// TwinCAT 3 PLC project StageCore
// Title: StageCore
// Company: _
// Author: Krystian Lis et al.
// ProjectVersion: 3.2.0
// ProgramVersion: 3.1.4026.16
// libraries:
//   Tc2_Math, * (Beckhoff Automation GmbH)
//   Tc2_Standard, * (Beckhoff Automation GmbH)
//   Tc2_System, * (Beckhoff Automation GmbH)
//   Tc2_Utilities, * (Beckhoff Automation GmbH)
// project tree:
//   Arg/Args/BOOL/ IArgToIBoolArg.TcPOU (not stored), BoolArg.TcPOU (not stored), I_BoolArg.TcIO (not stored)
//   Arg/Args/REAL/ IArgToIRealtArg.TcPOU (not stored), RealArg.TcPOU, I_RealArg.TcIO
//   Arg/Args/DWORD/ IArgToIDwordArg.TcPOU (not stored), DwordArg.TcPOU (not stored), I_DwordArg.TcIO
//   Arg/ ICompToIArg.TcPOU (not stored), IArgToIComp.TcPOU (not stored), I_Arg.TcIO (not stored)
//   Broadcast/Helpers/ GetSignal.TcPOU, GetReceiver.TcPOU (not stored)
//   Broadcast/Receiver/ AbstractReceiver.TcPOU (not stored), ICompToIRec.TcPOU, I_Receiver.TcIO, I_ReceiverNode.TcIO, Receiver.TcPOU (not stored)
//   Broadcast/Signal/ ICompToISignal.TcPOU, I_SignalEmit.TcIO (not stored), I_Signal.TcIO (not stored), I_SignalNode.TcIO, Signal.TcPOU (not stored)
//   Broadcast/Sys/Helpers/ _BroadcastDefragment.TcPOU, _BroadcastGetBestFit.TcPOU (not stored), _Emit.TcPOU, _Pair.TcPOU (not stored), _RegSignal.TcPOU (not stored), _Unpair.TcPOU
//   Broadcast/Sys/Structs/ _BroadcastStruct.TcDUT (not stored), _BroadcastUnion.TcDUT
//   Broadcast/Sys/ _Broadcast.TcGVL
//   Callable/ I_Callable.TcIO (not stored)
//   Dbg/ DebugInfo.TcPOU (not stored), DebugMsg.TcPOU, DebugStr.TcPOU (not stored), I_Debug.TcIO (not stored), _DebugInfo.TcDUT (not stored), _Debug.TcGVL (not stored)
//   Entity/Core/ Component.TcPOU, I_Component.TcIO, GetOwnerFromRaw.TcPOU, I_RawComponent.TcIO, I_Entity.TcIO (not stored), GetNextEntity.TcPOU, GetPrevEntity.TcPOU
//   Entity/Core/Scope/ EntityEnd.TcPOU (not stored), EntityExtend.TcPOU (not stored), EntityStart.TcPOU
//   Entity/Sys/ _EntityState.TcDUT, _Ec.TcGVL (not stored)
//   Entity/Sys/_Helpers/ _EntityEnd.TcPOU (not stored), _EntityExtend.TcPOU, _EntityStart.TcPOU, _RegisterComponent.TcPOU (not stored)
//   Entity/Sys/_Itf/ I_ComponentNode.TcIO (not stored), I_EntityNode.TcIO
//   Iter/ Iter.TcPOU
//   Result/Error/ Err.TcGVL, GenericResult.TcGVL (not stored)
//   Result/ IsErr.TcPOU (not stored), IsNone.TcPOU, IsOk.TcPOU (not stored), IsFail.TcPOU (not stored), IsSome.TcPOU (not stored), IsEnd.TcPOU, Result.TcDUT, ResultToStr.TcPOU
//   Runtime/Execute/ Execute.TcPOU (not stored), I_Execute.TcIO (not stored), I_ExecuteNode.TcIO
//   Runtime/Init/ Init.TcPOU, I_InitNode.TcIO, I_Init.TcIO (not stored)
//   Runtime/ Runtime.TcPOU, _Runtime.TcGVL (not stored)
//   State/_Buffer/ _StateBuffer.TcPOU (not stored)
//   State/Helpers/ GetStateManager.TcPOU, GetState.TcPOU
//   State/_Machine/ _StateMachine.TcPOU (not stored)
//   State/Manager/ ICompToIStateMgr.TcPOU (not stored), I_StateManager.TcIO, StateManager.TcPOU (not stored)
//   State/State/ ICompToIState.TcPOU, I_State.TcIO (not stored), I_StateInternal.TcIO (not stored), I_StateAdapter.TcIO (not stored), State.TcPOU (not stored)
//   Strings/Alias/ Ch.TcDUT, Str.TcDUT (not stored)
//   Strings/Strb/ I_Strb.TcIO (not stored), Strb.TcPOU (not stored)
//   Strings/Strf/ Strf.TcPOU (not stored)
//   Tags/Casts/ IArgToITag.TcPOU (not stored), ICompToITag.TcPOU, ICompToITagged.TcPOU
//   Tags/Helpers/ GetTag.TcPOU (not stored), GetTagOption.TcPOU, HasTagOption.TcPOU (not stored), HasTag.TcPOU, MatchPath.TcPOU
//   Tags/ I_Tag.TcIO, I_TagCmp.TcIO (not stored), I_Tagged.TcIO, TagBase.TcPOU (not stored), TagCmp.TcPOU, TagPath.TcPOU (not stored), Tag.TcPOU (not stored)
//   Tasks/Worker/Base/ Worker.TcPOU (not stored), I_Worker.TcIO
//   Tasks/Worker/ LoopWorker.TcPOU (not stored), BlockingWorker.TcPOU (not stored)
//   Tasks/TaskNode/ I_JobNode.TcIO, I_JobNodeInternal.TcIO, Job.TcPOU (not stored)
//   Tasks/ TaskState.TcDUT
//   Tasks/Job/ I_Job.TcIO (not stored)
//   _/ Param.TcGVL
// (motion and I/O tree: see PLC project stageutils)
// real-time tasks:
//   TASK Example: cycle T#10ms, priority 20, ADS port 350
//   TASK Test: cycle T#10ms, priority 21, ADS port 351
//   TASK VISU_TASK: cycle T#200000us, priority 30, ADS port 352

// ---- Broadcast/Sys/Structs/_BroadcastUnion.TcDUT
TYPE INTERNAL  _BroadcastUnion :
UNION
	iSignal		: I_SignalNode;
	iReceiver	: I_ReceiverNode;
END_UNION
END_TYPE

// ---- Entity/Sys/_EntityState.TcDUT
{attribute 'qualified_only'}
{attribute 'strict'}
TYPE INTERNAL _EntityState :
(
	Unregistered,
	Registered,
	Completed
);
END_TYPE

// ---- Result/Result.TcDUT
// Alias for INT values.
// | Result >= 1 - Ok/Success
// | Result = 0 - None
// | Result <=- 1 - Error
TYPE Result : INT; END_TYPE

// ---- Strings/Alias/Ch.TcDUT
// Alias for STRING(1) values.
TYPE Ch : STRING(1); END_TYPE

// ---- Tasks/TaskState.TcDUT
{attribute 'qualified_only'}
{attribute 'strict'}
TYPE TaskState :
(
	Error,
	Idle,
	Ready,
	Running,
	Aborted,
	Completed
) BYTE := Idle;
END_TYPE

// ---- Broadcast/Sys/_Broadcast.TcGVL
{attribute 'qualified_only'}
VAR_GLOBAL INTERNAL
	{attribute 'ExpandFully'} 
	entry				: ARRAY[1..Param.RECEIVER_CAP] OF _BroadcastStruct;
	iSignal				: ARRAY[1..Param.SIGNAL_CAP] OF I_SignalNode;
	iFirst				: I_SignalNode;
	nRecLen				: UDINT;
	nSignalLen			: UDINT;
END_VAR

// ---- Result/Error/Err.TcGVL
{attribute 'qualified_only'}
VAR_GLOBAL CONSTANT
	Itf0			: Result := -2; // Null Interface 
	Str0			: Result := -3; // Empty String
	ItfEq			: Result := -4; // Interfaces are equal
	NoMatch			: Result := -5; // No match
	Ptr0			: Result := -6; // Null Pointer
	InvRef			: Result := -7; // Invalid reference
	Ovf				: Result := -8; // Overflow/Out of bounds
	Udf				: Result := -9; // Undefined
	Idx				: Result := -10; // Index error
	TcLib			: Result := -11; // Error caused by TwinCAT libraries
	InfLoop			: Result := -12; // Potential infinity loop
	IncArg			: Result := -13; // Incorrect input argument
	Init			: Result := -14; // Initialisation error
	NotFound		: Result := -15; // Item not found
	InvItf			: Result := -16; // Invalid interface
	End				: Result := -17; // End of collection
END_VAR

// ---- _/Param.TcGVL
{attribute 'qualified_only'}
// DO NOT SET ANY OF THE CAP PARAMETERS TO 0 OR LARGER THAN MAX DINT!!!
VAR_GLOBAL CONSTANT
	DEBUGMSG_CAP	: UDINT(1..16#7FFFFFFF) := 10; // Max number of debug messages.
	DEBUGSTR_CAP	: UDINT(1..16#7FFFFFFF) := 500; // Max number of debug strings.
	
	SIGNAL_CAP		: UDINT(1..16#7FFFFFFF) := 20; // Max number of signals.
	RECEIVER_CAP	: UDINT(1..16#7FFFFFFF) := 100; // Max number of signal-receiver pairings.
END_VAR

// ---- Arg/Args/REAL/I_RealArg.TcIO
(*
A broadcastable wrapper for a `REAL` value. 
*)
INTERFACE I_RealArg EXTENDS I_Arg

(*
Reads the internal value.
*)
PROPERTY Get : REAL
GET
END_GET
END_PROPERTY

(*
Returns TRUE if the value is mutable.
*)
PROPERTY IsMut : BOOL
GET
END_GET
END_PROPERTY

(*
Modifies the internal value.  
Returns:
- `Ok` - Upon successful modification.
- `Error` - If mutability is disabled.
*)
METHOD Set : Result
VAR_INPUT
	newVal		: REAL;
END_VAR
END_METHOD

END_INTERFACE

// ---- Arg/Args/DWORD/I_DwordArg.TcIO
(*
A broadcastable wrapper for a `DWORD` value. 
*)
INTERFACE I_DwordArg EXTENDS I_Arg

(*
Reads the internal value.
*)
PROPERTY Get : DWORD
GET
END_GET
END_PROPERTY

(*
Returns TRUE if the value is mutable.
*)
PROPERTY IsMut : BOOL
GET
END_GET
END_PROPERTY

(*
Modifies the internal value.  
Returns:
- `Ok` - Upon successful modification.
- `Error` - If mutability is disabled.
*)
METHOD Set : Result
VAR_INPUT
	newVal		: DWORD;
END_VAR
END_METHOD

END_INTERFACE

// ---- Broadcast/Receiver/I_Receiver.TcIO
(*
Represents a receiver in the Broadcast system. Implements the necessary methods for receiving events and pairing signals.
Can be casted to `I_Component`.
*)
INTERFACE I_Receiver EXTENDS I_ReceiverNode, I_Tagged

END_INTERFACE

// ---- Broadcast/Receiver/I_ReceiverNode.TcIO
INTERFACE INTERNAL I_ReceiverNode EXTENDS I_Debug

METHOD INTERNAL Receive
VAR_INPUT
	iArg			: I_Arg;
END_VAR
END_METHOD

END_INTERFACE

// ---- Broadcast/Signal/I_SignalNode.TcIO
INTERFACE INTERNAL I_SignalNode EXTENDS I_Debug

PROPERTY INTERNAL _End : UDINT
GET
END_GET
SET
END_SET
END_PROPERTY

PROPERTY INTERNAL _Id : UDINT
GET
END_GET
END_PROPERTY

PROPERTY INTERNAL _Size : UDINT
GET
END_GET
SET
END_SET
END_PROPERTY

PROPERTY INTERNAL _Start : UDINT
GET
END_GET
SET
END_SET
END_PROPERTY

END_INTERFACE

// ---- Entity/Core/I_Component.TcIO
(*
Stores raw I_RawComponent value and additional metadata.
*)
INTERFACE I_Component EXTENDS I_ComponentNode

(*
Returns parent Entity.
*)
PROPERTY Entity : I_Entity
GET
END_GET
END_PROPERTY

(*
Returns raw I_RawComponent pointer.
*)
PROPERTY Raw : I_RawComponent
GET
END_GET
END_PROPERTY

END_INTERFACE

// ---- Entity/Core/I_RawComponent.TcIO
(*
Represents a component in the Entity-Component system.  
Can be cast to other interfaces for extended functionality and interaction.
*)
INTERFACE I_RawComponent EXTENDS __SYSTEM.IQueryInterface, I_Debug

END_INTERFACE

// ---- Entity/Sys/_Itf/I_EntityNode.TcIO
INTERFACE INTERNAL I_EntityNode EXTENDS I_Debug

PROPERTY INTERNAL _AsIEntity : I_Entity
GET
END_GET
END_PROPERTY

PROPERTY INTERNAL _FirstComp : I_ComponentNode
GET
END_GET
SET
END_SET
END_PROPERTY

PROPERTY INTERNAL _LastComp : I_ComponentNode
GET
END_GET
SET
END_SET
END_PROPERTY

PROPERTY INTERNAL _Next : I_EntityNode
GET
END_GET
SET
END_SET
END_PROPERTY

PROPERTY INTERNAL _Prev : I_EntityNode
GET
END_GET
SET
END_SET
END_PROPERTY

PROPERTY INTERNAL _Size : UDINT
GET
END_GET
SET
END_SET
END_PROPERTY

PROPERTY INTERNAL _State : _EntityState
GET
END_GET
SET
END_SET
END_PROPERTY

(*
Description: Retrieves a previous component before the inputted one or last component if referenced value is 0.
Returns:
- Ok - Returns upon success, updates referenced value with new component.
- Err.InvRef - Invalid output reference.
- Err.ItfEq - Provided interface pointer doesn't belong to the queried entity. Nulls reference.
- Err.NotFound - The entity doesn't contain any components. Nulls reference.
- Err.End - No more components. Nulls reference.
*)
METHOD GetNextComp : Result
VAR_INPUT
	iOut		: REFERENCE TO I_Component;
END_VAR
END_METHOD

(*
Description: Retrieves a previous component before the inputted one or last component if referenced value is 0.
Returns:
- Ok - Returns upon success, updates referenced value with new component.
- Err.InvRef - Invalid output reference.
- Err.ItfEq - Provided interface pointer doesn't belong to the queried entity. Nulls reference.
- Err.NotFound - The entity doesn't contain any components. Nulls reference.
- Err.End - No more components. Nulls reference.
*)
METHOD GetPrevComp : Result
VAR_INPUT
	iOut		: REFERENCE TO I_Component;
END_VAR
END_METHOD

(*
Provides the size of the entity, indicating the number of components it manages.  
Note: For internal logic purposes, this value is incremented by one beyond the actual component count.
*)
PROPERTY Size : UDINT
GET
END_GET
END_PROPERTY

END_INTERFACE

// ---- Runtime/Execute/I_ExecuteNode.TcIO
INTERFACE INTERNAL I_ExecuteNode EXTENDS I_Debug;

METHOD INTERNAL Attach : Result
VAR_INPUT
	iExecute		: I_ExecuteNode;
END_VAR
END_METHOD

METHOD INTERNAL Exe
VAR_OUTPUT
	iNext: I_ExecuteNode;
END_VAR
END_METHOD

PROPERTY INTERNAL State : Result
GET
END_GET
SET
END_SET
END_PROPERTY

END_INTERFACE

// ---- Runtime/Init/I_InitNode.TcIO
INTERFACE INTERNAL I_InitNode EXTENDS I_Debug;

METHOD INTERNAL Attach : Result
VAR_INPUT
	iInit		: I_InitNode;
END_VAR
END_METHOD

METHOD INTERNAL Init
VAR_OUTPUT
	iNext: I_InitNode;
END_VAR
END_METHOD

PROPERTY INTERNAL State : Result
GET
END_GET
SET
END_SET
END_PROPERTY

END_INTERFACE

// ---- State/Manager/I_StateManager.TcIO
(*
Can be casted to `I_Component`.
Manages the lifecycle and transitions of states within an entity.  
Supports queuing state change requests, triggering state transitions, and broadcasting state change events.  
Adds a `_stateChangeEvent` Signal to the owning `I_Entity` during initialization, enabling external components to listen for state changes.
*)
INTERFACE I_StateManager EXTENDS I_Debug, I_RawComponent

(*
Retrieves the currently active state managed by the state manager.
*)
PROPERTY Current : I_State
GET
END_GET
END_PROPERTY

(*
Returns the entity that owns this state.
*)
PROPERTY Owner : I_Entity
GET
END_GET
END_PROPERTY

(*
Retrieves the state that is queued to become active next, but has not yet transitioned.
*)
PROPERTY Pretender : I_State
GET
END_GET
END_PROPERTY

(*
Retrieves the last active state prior to the current one.
*)
PROPERTY Previous : I_State
GET
END_GET
END_PROPERTY

(*
Queues a request to transition to a specified state.  

Returns:
- `Ok` - If the state change request is successfully queued.
- `Err.Itf0` - If the provided state interface is invalid.
- `Err.NoMatch` - If the state does not belong to the same entity.
- `Err.IncArg` - If the state is already in the queue.
*)
METHOD Request : Result
VAR_INPUT
	iState		: I_State;
END_VAR
END_METHOD

END_INTERFACE

// ---- Tags/I_Tag.TcIO
(*
An identifier that uses reflection to generate a unique symbol path.
It simplifies the path by removing project, PLC, and tag segments.
Can be casted to `I_Arg` and `I_Component`.
Example:
- Reflection: proj.plc.MAIN.functionBlock[*]._tag
- Path: MAIN.functionBlock.5
*)
INTERFACE I_Tag EXTENDS I_Debug, I_Component, I_Arg

// Read address path without Option segment.
PROPERTY Id : Str
GET
END_GET
END_PROPERTY

// Modify or read the optional segment.
PROPERTY Option : Str
GET
END_GET
END_PROPERTY

END_INTERFACE

// ---- Tags/I_Tagged.TcIO
(*
This component contains readable `I_Tag`.
Can be casted to `I_Component`.
*)
INTERFACE I_Tagged EXTENDS I_RawComponent

PROPERTY Tag : I_Tag
GET
END_GET
END_PROPERTY

END_INTERFACE

// ---- Tasks/Worker/Base/I_Worker.TcIO
INTERFACE I_Worker EXTENDS I_Debug

METHOD Defer : Result
VAR_INPUT
    iJob : I_JobNode;
END_VAR
END_METHOD

METHOD Dequeue : Result
VAR_INPUT
	iJob: I_JobNode;
END_VAR
END_METHOD

METHOD Enqueue : Result
VAR_INPUT
	iJob: I_JobNode;
END_VAR
END_METHOD

PROPERTY First : I_JobNode
GET
END_GET
END_PROPERTY

END_INTERFACE

// ---- Tasks/TaskNode/I_JobNode.TcIO
INTERFACE I_JobNode EXTENDS I_JobNodeInternal

END_INTERFACE

// ---- Tasks/TaskNode/I_JobNodeInternal.TcIO
INTERFACE INTERNAL I_JobNodeInternal EXTENDS I_Debug

PROPERTY INTERNAL _Next : I_JobNode
GET
END_GET
SET
END_SET
END_PROPERTY

PROPERTY INTERNAL _Prev : I_JobNode
GET
END_GET
SET
END_SET
END_PROPERTY

METHOD INTERNAL _Reset
VAR_INPUT
END_VAR
END_METHOD

METHOD INTERNAL _Run
VAR_INPUT
END_VAR
END_METHOD

PROPERTY State : TaskState
GET
END_GET
END_PROPERTY

PROPERTY Worker : I_Worker
GET
END_GET
END_PROPERTY

END_INTERFACE

// ---- Runtime/Init/Init.TcPOU
(*
Allows registration of FB implementing `I_Init`. 
*)
FUNCTION_BLOCK FINAL Init IMPLEMENTS I_InitNode, I_Debug
VAR
	_iInit			: I_Init;
	_iNext			: I_InitNode;
	_nState			: Result;
	_nPhase			: INT;
END_VAR

METHOD INTERNAL Attach : Result
VAR_INPUT
	iInit			: I_InitNode;
END_VAR
VAR
	_iThis			: I_InitNode := THIS^;
END_VAR
IF iInit = 0 THEN
	DebugMsg(0, Tc2_Standard.CONCAT(__POUNAME(), ': Itf = 0!'));
	RETURN;
END_IF

IF _iThis <> _Runtime.iLastInit THEN
	DebugMsg(THIS^, Tc2_Standard.CONCAT(__POUNAME(), ': Is not the last node!'));
	RETURN;
END_IF

IF IsSome(iInit.state) THEN
	DebugMsg(iInit, Tc2_Standard.CONCAT(__POUNAME(), ': Has already been added!'));
	RETURN;
END_IF

_Runtime.iLastInit := iInit;
_iNext := iInit;
END_METHOD

//FB_Init is always available implicitly and it is used primarily for initialization.
//The return value is not evaluated. For a specific influence, you can also declare the
//methods explicitly and provide additional code there with the standard initialization
//code. You can evaluate the return value.
{attribute 'hide'}
METHOD FB_Init: BOOL
VAR_INPUT
    bInitRetains: BOOL; // TRUE: the retain variables are initialized (reset warm / reset cold)
    bInCopyCode: BOOL;  // TRUE: the instance will be copied to the copy code afterward (online change)
	
	iInit			: I_Init;
END_VAR
IF IsSome(_nState) THEN
	RETURN;
END_IF

IF (_iInit := iInit) = 0 THEN
	_nState := Err.Itf0;
	DebugMsg(THIS^, Tc2_Standard.CONCAT(__POUNAME(), ': Itf = 0!'));
	RETURN;
END_IF



IF _Runtime.iLastInit <> 0 THEN
	IF IsErr(_Runtime.iLastInit.Attach(THIS^), nOut => _nState) THEN
		DebugMsg(THIS^, Tc2_Standard.CONCAT(__POUNAME(), ': Error Inside!'));
	END_IF
ELSE
	_Runtime.iFirstInit := THIS^;
	_Runtime.iLastInit := THIS^;
	_nState := Ok;
END_IF
END_METHOD

METHOD INTERNAL Init
VAR_OUTPUT
	iNext: I_InitNode;
END_VAR
_iInit.Init(_nPhase);
iNext := _iNext;
END_METHOD

PROPERTY Phase : INT
GET
Phase := _nPhase;
END_GET
SET
_nPhase := Phase;
END_SET
END_PROPERTY

PROPERTY INTERNAL State : Result
GET
State := _nState;
END_GET
SET
IF IsNone(_nState) THEN
	_nState := State;
END_IF
END_SET
END_PROPERTY

END_FUNCTION_BLOCK

// ---- Dbg/DebugMsg.TcPOU
(*
Logs a debug message as a string tied to a `I_Debug` interface for inspection and troubleshooting within the IDE.
*)
FUNCTION DebugMsg
VAR_INPUT
	iDebug			: I_Debug;
	sInfo			: Str;
END_VAR

_Debug.nErrorNumber := _Debug.nErrorNumber + 1;

IF _Debug.nLastMsg < Param.DEBUGMSG_CAP THEN
	_Debug.nLastMsg := _Debug.nLastMsg + 1;
ELSE
	_Debug.nLastMsg := 1;
END_IF

_Debug.debugMsg[_Debug.nLastMsg].iDebug := iDebug;
_Debug.debugMsg[_Debug.nLastMsg].sInfo := sInfo;

END_FUNCTION

// ---- Result/IsNone.TcPOU
// Return TRUE if the value is None.
// Optionally carries the value over to nOut for further processing.
FUNCTION IsNone : BOOL
VAR_INPUT
    nIn : Result; // Result variable to check for None
END_VAR
VAR_OUTPUT
    nOut : Result; // Carries the input value for further use
END_VAR

IsNone := nIn = 0;
nOut := nIn;

END_FUNCTION

// ---- Arg/Args/REAL/RealArg.TcPOU
(*
A broadcastable wrapper for a `REAL` value. 
*)
FUNCTION_BLOCK RealArg IMPLEMENTS I_RealArg
VAR
	_val			: REAL;
	_bMut			: BOOL := FALSE;
END_VAR

(*
Enables external modification of the internal value.
*)
METHOD AllowMut
_bMut := TRUE;
END_METHOD

(*
Disables external modification of the internal value.
*)
METHOD BlockMut
_bMut := FALSE;
END_METHOD

//FB_Init is always available implicitly and it is used primarily for initialization.
//The return value is not evaluated. For a specific influence, you can also declare the
//methods explicitly and provide additional code there with the standard initialization
//code. You can evaluate the return value.
{attribute 'hide'}
METHOD FB_Init: BOOL
VAR_INPUT
    bInitRetains: BOOL; // TRUE: the retain variables are initialized (reset warm / reset cold)
    bInCopyCode: BOOL;  // TRUE: the instance will be copied to the copy code afterward (online change)   

	initVal		: REAL;
END_VAR
_val := initVal;
END_METHOD

(*
Reads the internal value.
*)
PROPERTY Get : REAL
GET
Get := _val;
END_GET
END_PROPERTY

(*
Returns TRUE if the value is mutable.
*)
PROPERTY IsMut : BOOL
GET
IsMut := _bMut;
END_GET
END_PROPERTY

(*
Directly modifies the internal value, bypassing any mutability restrictions.
*)
METHOD OpSet : I_Arg
VAR_INPUT
	newVal		: REAL;
END_VAR
_val := newVal;
OpSet := THIS^;
END_METHOD

(*
Modifies the internal value.  
Returns:
- `Ok` - Upon successful modification.
- `Error` - If mutability is disabled.
*)
METHOD Set : Result
VAR_INPUT
	newVal		: REAL;
END_VAR
IF _bMut THEN
	_val := newVal;
	Set := Ok;
ELSE
	Set := Error;
END_IF
END_METHOD

END_FUNCTION_BLOCK

// ---- Broadcast/Helpers/GetSignal.TcPOU
(*
Searches an `I_Entity` for a `I_Signal` component matching provided id pattern.
Result:
- Ok - Returns `I_Signal`.
- Err.NotFound - Returns null.
- Err.InvRef - Returns null.
- Err.Itf0 - Returns null, incorrect interface.
*)
FUNCTION GetSignal : Result
VAR_INPUT
	iEntity		: I_Entity;
	sTagId		: Str;
	iOut		: REFERENCE TO I_Signal;
END_VAR
VAR
	_iComp		: I_Component;
	cmp			: TagCmp;
END_VAR

IF iEntity = 0 THEN
	GetSignal := Err.Itf0;
	RETURN;
END_IF

IF NOT __ISVALIDREF(iOut) THEN
	GetSignal := Err.InvRef;
	RETURN;
END_IF

WHILE IsOk(iEntity.GetNextComp(_iComp)) DO
	IF IsOk(ICompToISignal(_iComp.Raw, iOut)) THEN
		IF cmp.Set(iOut.Tag).MatchWcdId(sTagId).IsTrue() THEN
			GetSignal := Ok;
			RETURN;
		ELSE
			iOut := 0;
		END_IF
	END_IF
END_WHILE

GetSignal := Err.NotFound;

END_FUNCTION

// ---- Tags/TagCmp.TcPOU
(*
A tool for performing CASE OF-like evaluations on `I_Tag`.  
It enables sequential evaluation of conditions and stops when `IsTrue`, `IsFalse`, or `IsErr` methods are invoked.
Allows method chaining.
*)
FUNCTION_BLOCK FINAL TagCmp IMPLEMENTS I_TagCmp
VAR
	_iBaseTag		: I_Tag;
	_nResult		: Result;
	_bLock			: BOOL;
END_VAR

PROPERTY PRIVATE _self : I_TagCmp
GET
VAR
	_this : I_TagCmp := THIS^;
END_VAR
_self := _this;
END_GET
END_PROPERTY

(*
Updates its internal state based on the internal status and option.  
Sets the state to `Ok` if the base tag is `Ok` and has the specified Option; otherwise, sets the state to `None`.
*)
METHOD AndHasOption : I_TagCmp

VAR_INPUT
	sOption		: Str;
END_VAR
AndHasOption := _self;
sOption := Tc2_Utilities.F_ToLCase(sOption);

IF _bLock THEN
	RETURN;
END_IF

IF _nResult = Ok AND _iBaseTag.Option = sOption THEN
	_nResult := Ok;
ELSE
	_nResult := None;
END_IF
END_METHOD

(*
Updates its internal state based on the internal status and an external condition.  
Sets the state to `Ok` if the base tag is `Ok` and the external condition is TRUE; otherwise, sets the state to `None`.
*)
METHOD AndIf : I_TagCmp
VAR_INPUT
	bCondition: BOOL;
END_VAR
AndIf := _self;

IF _bLock THEN
	RETURN;
END_IF

IF _nResult = Ok AND_THEN bCondition THEN
	_nResult := Ok;
ELSE
	_nResult := None;
END_IF
END_METHOD

(*
Updates its internal state based on the internal status and option.  
Sets the state to `Ok` if the base tag has the specified Option.
*)
METHOD HasOption : I_TagCmp
VAR_INPUT
	sOption		: Str;
END_VAR
HasOption := _self;
sOption := Tc2_Utilities.F_ToLCase(sOption);

IF _bLock THEN
	RETURN;
END_IF

CASE _nResult OF
	Ok,
	None:
		IF sOption <> '' AND_THEN _iBaseTag.Option = sOption THEN
			_nResult := Ok;
		END_IF
END_CASE
END_METHOD

(*
Returns `TRUE` if any evaluated conditions resulted in `Error`.  
Halts further evaluations by locking the current state.
*)
METHOD IsErr : BOOL
VAR_INPUT
END_VAR
IF _bLock THEN
	RETURN;
END_IF

IF _nResult >= 0 THEN
	RETURN;
END_IF

_bLock := TRUE;
IsErr := TRUE;
END_METHOD

(*
Returns `TRUE` if all evaluated conditions resulted in `FALSE`.  
Halts further evaluations by locking the current state.
*)
METHOD IsFalse : BOOL
VAR_INPUT
END_VAR
IF _bLock THEN
	RETURN;
END_IF

IF _nResult <> None THEN
	RETURN;
END_IF

_bLock := TRUE;
IsFalse := TRUE;
END_METHOD

(*
Returns `TRUE` if any evaluated condition resulted in `TRUE`.  
Halts further evaluations by locking the current state.
*)
METHOD IsTrue : BOOL
VAR_INPUT
END_VAR
IF _bLock THEN
	RETURN;
END_IF

IF _nResult <> Ok THEN
	RETURN;
END_IF

_bLock := TRUE;
IsTrue := TRUE;
END_METHOD

(*
Updates its internal state based on the internal status and external I_Tag.  
Sets the state to `Ok` if the base tag matches the external tag.
*)
METHOD Match : I_TagCmp
VAR_INPUT
	iOther: I_Tag;
END_VAR
Match := _self;

IF _bLock THEN
	RETURN;
END_IF

CASE _nResult OF
	Ok,
	None:
		IF iOther = _iBaseTag THEN
			_nResult := Ok;
		END_IF
END_CASE
END_METHOD

(*
Updates its internal state based on the internal status and a string value.  
Sets the state to `Ok` if the base tag Id matches the provided string from right to left.
*)
METHOD MatchId : I_TagCmp
VAR_INPUT
	sIdToMatch		: Str;
END_VAR
MatchId := _self;
sIdToMatch := Tc2_Utilities.F_ToLCase(sIdToMatch);

IF _bLock THEN
	RETURN;
END_IF

CASE _nResult OF
	Ok,
	None:
		IF sIdToMatch <> '' AND_THEN (Tc2_Standard.RIGHT(_iBaseTag.Id, Tc2_Standard.LEN(sIdToMatch)) = sIdToMatch) THEN
			_nResult := Ok;
		END_IF
END_CASE
END_METHOD

(*
Updates its internal state based on the internal status and a string value.  
Sets the state to `Ok` if the base tag Id matches the provided string pattern.
Allows wildcards.
*)
METHOD MatchWcdId : I_TagCmp
VAR_INPUT
	sPattern 			: Str;
END_VAR
VAR
	pttPath				: TagPath;
	pttSeg				: Str;
	pttPeek				: Str;
	addPath				: TagPath;
	addSeg				: Str;
	bMatch				: BOOL;
END_VAR
MatchWcdId := _self;

// Check lock
IF _bLock THEN
	RETURN;
END_IF

// Check result state
CASE _nResult OF
	Ok,
	None:		
		_nResult := MatchPath(_iBaseTag.Id, sPattern);
END_CASE
END_METHOD

(*
Updates its internal state based on the internal status and an external condition.  
Sets the state to `Ok` if the base tag is `Ok` or the external condition is TRUE.
*)
METHOD OrIf : I_TagCmp
VAR_INPUT
	bCondition: BOOL;
END_VAR
OrIf := _self;

IF _bLock THEN
	RETURN;
END_IF

IF _nResult = Ok OR_ELSE bCondition THEN
	_nResult := Ok;
END_IF
END_METHOD

(*
Sets a new base tag for comparison and resets the result and lock states.
Fails if `iBaseTag` is `0`;
*)
METHOD Set : I_TagCmp
VAR_INPUT
	iBaseTag	: I_Tag;
END_VAR
_iBaseTag := iBaseTag;
_nResult := None;
_bLock := FALSE;

IF iBaseTag = 0 THEN
	_nResult := Err.Itf0;
END_IF

Set := _self;
END_METHOD

(*
Updates its internal state based on the internal status and an external condition.  
Sets the state to `Ok` if the base tag is `Ok` xor the external condition is TRUE.
*)
METHOD XorIf : I_TagCmp
VAR_INPUT
	bCondition: BOOL;
END_VAR
XorIf := _self;

IF _bLock THEN
	RETURN;
END_IF

IF _nResult = Ok XOR bCondition THEN
	_nResult := Ok;
END_IF
END_METHOD

END_FUNCTION_BLOCK

// ---- Tags/Helpers/MatchPath.TcPOU
(*
Returns whether the symbol's path matches the provided pattern.
Allows wildcards in form of "*" that can cover multiple segments.
Example pattern: *.functionBlock.*.bBool
*)
FUNCTION MatchPath : Result
VAR_INPUT
    sAddress : Str;  /// The symbol's path to evaluate
    sPattern : Str;  /// The pattern to match against
END_VAR
VAR
	pttPath				: TagPath;
	pttSeg				: Str;
	pttPeek				: Str;
	addPath				: TagPath;
	addSeg				: Str;
	bMatch				: BOOL;
END_VAR

// Init
IF IsErr(addPath.Set(sAddress)) THEN
	MatchPath := Err.NoMatch;
	RETURN;
END_IF
IF IsErr(pttPath.Set(sPattern)) THEN
	MatchPath := Err.NoMatch;
	RETURN;
END_IF

// Advance to the next segment
WHILE IsOk(pttPath.Next(sSeg => pttSeg)) DO	
	bMatch := FALSE;
	// If the current segment is a wildcard, then peek to the next segment
	IF pttSeg = '*' THEN
		IF IsOk(pttPath.Peek(sSeg => pttPeek)) THEN
			IF pttPeek = '*' THEN
				CONTINUE; // Skip redundant wildcard if *.*.
			END_IF
		ELSE
			MatchPath := Ok;
			RETURN; // No more segments in the pattern, so it's a match as everything so far matched(.*)
		END_IF

	// If current segment is not a wildcard reset the peek.
	ELSIF pttSeg <> '*' THEN
		pttPeek := '';
	END_IF
	
	// Get the next segment of the address path
	WHILE IsOk(addPath.Next(sSeg => addSeg)) DO
		IF pttPeek <> '' THEN
			IF pttPeek = addSeg THEN
				bMatch := TRUE;
				pttPath.Next(); // Consume get next pattern segment
				EXIT;
			ELSE
				CONTINUE; // Get next address
			END_IF
		ELSIF pttSeg = addSeg THEN
			bMatch := TRUE;
			EXIT; // Consume get next pattern segment
		ELSE
			MatchPath := Err.NoMatch;
			RETURN; // No match - return
		END_IF
	END_WHILE

	IF NOT bMatch THEN
		MatchPath := Err.NoMatch;
		RETURN;
	END_IF

END_WHILE

IF IsOk(addPath.Peek()) THEN
	MatchPath := Err.NoMatch;
	RETURN;
END_IF

MatchPath := Ok;

END_FUNCTION

// ---- Broadcast/Signal/ICompToISignal.TcPOU
(*
Casts I_Component as I_Signal.
Returns:
- Ok - Success,
- Err.InvRef - Invalid reference,
- Err.Itf0 - Invalid interface,
- Err.NoMatch - Cast failed
*)
FUNCTION ICompToISignal : Result
VAR_INPUT
	iIn	: I_Component;
	iOut: REFERENCE TO I_Signal;
END_VAR

IF NOT __ISVALIDREF(iOut) THEN
	ICompToISignal := Err.InvRef;
	RETURN;
END_IF

IF iIn = 0 THEN
	ICompToISignal := Err.Itf0;
	RETURN;
END_IF

IF __QUERYINTERFACE(iIn, iOut) THEN
	ICompToISignal := Ok;
ELSE
	ICompToISignal := Err.NoMatch;
END_IF

END_FUNCTION

// ---- Broadcast/Receiver/ICompToIRec.TcPOU
(*
Casts I_Component as I_Receiver.
Returns:
- Ok - Success,
- Err.InvRef - Invalid reference,
- Err.Itf0 - Invalid interface,
- Err.NoMatch - Cast failed
*)
FUNCTION ICompToIRec : Result
VAR_INPUT
	iIn		: I_RawComponent;
	iOut	: REFERENCE TO I_Receiver;
END_VAR

IF NOT __ISVALIDREF(iOut) THEN
	ICompToIRec := Err.InvRef;
	RETURN;
END_IF

IF iIn = 0 THEN
	ICompToIRec := Err.Itf0;
	RETURN;
END_IF

IF __QUERYINTERFACE(iIn, iOut) THEN
	ICompToIRec := Ok;
ELSE
	ICompToIRec := Err.NoMatch;
END_IF

END_FUNCTION

// ---- Broadcast/Sys/Helpers/_BroadcastDefragment.TcPOU
FUNCTION INTERNAL _BroadcastDefragment : Result
VAR_INPUT
	iLastSignal		: I_SignalNode := 0;
END_VAR
VAR
	i				: UDINT;
   _temp			: ARRAY[1..Param.RECEIVER_CAP] OF _BroadcastStruct;
   _iSwappedSignal	: I_SignalNode;
   _nNextCopyId		: UDINT := 1;
END_VAR

// 1) If we are at maximum capacity (all slots are allocated).
IF _Broadcast.nRecLen = Param.RECEIVER_CAP THEN
    _BroadcastDefragment := Err.Ovf;
    RETURN;
END_IF

// 2) If there are no allocated slots at all, nothing to defragment.
IF _Broadcast.nRecLen = 0 THEN
    _BroadcastDefragment := Ok;
    RETURN;
END_IF

// 3) We want to ensure that entity that requires more space will get it, so we move it temporarly to the end.
IF iLastSignal <> 0 THEN
	_iSwappedSignal := _Broadcast.iSignal[_Broadcast.nSignalLen];
	_Broadcast.iSignal[iLastSignal._Id] := _iSwappedSignal;
	_Broadcast.iSignal[_Broadcast.nSignalLen] := iLastSignal;
END_IF

// 3) Copy all chunks to the temporary table
FOR i := 1 TO _Broadcast.nSignalLen DO
	IF _Broadcast.iSignal[i]._Start <> 0 THEN
		Tc2_SYSTEM.MEMCPY(
							ADR(_temp[_nNextCopyId]),
							ADR(_Broadcast.entry[_Broadcast.iSignal[i]._Start]),
							SIZEOF(_EcStruct) * _Broadcast.iSignal[i]._Size
						);
		_Broadcast.iSignal[i]._Start := _nNextCopyId;
		_nNextCopyId := _Broadcast.iSignal[i]._Size + _nNextCopyId;
		_Broadcast.iSignal[i]._End := _nNextCopyId - 1;	
	END_IF
END_FOR

// 3) Move back the swapped entities, to preserve the Ids.
IF iLastSignal <> 0 THEN
	_Broadcast.iSignal[_iSwappedSignal._Id] := _iSwappedSignal;
	_Broadcast.iSignal[iLastSignal._Id] := iLastSignal;
END_IF

// 4) Copy temporary table onto the _Ec.comp table
Tc2_System.MEMCPY(
	ADR(_Broadcast.entry),
	ADR(_temp),
	SIZEOF(_EcStruct) * _Broadcast.nRecLen
);

// 5) Clear the remainging area
Tc2_System.MEMSET(
	ADR(_Broadcast.entry[_Broadcast.nRecLen + 1]),
	0,
	SIZEOF(_EcStruct) * (Param.RECEIVER_CAP - _Broadcast.nRecLen)
);

// 6) First entry in _Ec.comp should always be iFirst
CASE _Broadcast.entry[1].nType OF
	1:
		_BroadcastDefragment := Ok;
		_Broadcast.iFirst := _Broadcast.entry[1].variant.iSignal;
	ELSE
		_BroadcastDefragment := Err.Udf;
END_CASE

END_FUNCTION

// ---- Broadcast/Sys/Helpers/_Emit.TcPOU
FUNCTION INTERNAL _Emit : Result
VAR_INPUT
	iSignal		: I_SignalNode;
	iArg		: I_Arg;
END_VAR
VAR
	i			: UDINT;
	_nEnd		: UDINT;
END_VAR

IF iSignal = 0 THEN
	RETURN;
END_IF

IF iSignal._Start = 0 THEN
	RETURN;
END_IF

_nEnd := iSignal._End;
// Assumes that the entry table is correctly constructed which is very likely
FOR i := iSignal._Start + 1 TO _nEnd DO
	_Broadcast.entry[i].variant.iReceiver.Receive(iArg);
END_FOR

END_FUNCTION

// ---- Broadcast/Sys/Helpers/_Unpair.TcPOU
FUNCTION INTERNAL _Unpair : Result
VAR_INPUT
	iSignal		: I_SignalNode;
	iReceiver	: I_ReceiverNode;
END_VAR
VAR
	i			: UDINT;
	_nPos		: UDINT;
	_nEnd		: UDINT;
	_nFirstId	: UDINT := Param.RECEIVER_CAP;
	_nNewStart	: UDINT;
END_VAR

// 1) Basic null check
IF iSignal = 0 OR iReceiver = 0 THEN
	_Unpair := Err.Itf0;
	RETURN;
END_IF

// 2) Find iReceiver in [iSignal._Start+1 .. iSignal._End]
_nEnd := iSignal._End;
FOR i := iSignal._Start + 1 TO _nEnd DO
	IF _Broadcast.entry[i].variant.iReceiver = iReceiver THEN
		_nPos := i;
		EXIT;
	END_IF
END_FOR

// 3) If not found, return an error
IF _nPos = 0 THEN
	_Unpair := Err.NoMatch;
	RETURN;
END_IF

// 4) Decrement the signal's size (removing one receiver)
iSignal._Size := iSignal._Size - 1;

// 5) If only the header slot remains, remove the signal entirely
IF iSignal._Size = 1 THEN
	// Clear the last receiver slot
	_Broadcast.entry[_nEnd].nType := 0;
	_Broadcast.entry[_nEnd].variant.iReceiver := 0;
	// Clear the signal header slot
	_Broadcast.entry[_nEnd - 1].nType := 0;
	_Broadcast.entry[_nEnd - 1].variant.iSignal := 0;
	// Reset iSignal metadata
	iSignal._Size := 0;
	iSignal._Start := 0;
	iSignal._End := 0;

	// If this was the leftmost signal, find a new one
	IF _Broadcast.iFirst = iSignal THEN
		FOR i := 1 TO _Broadcast.nSignalLen DO
			_nNewStart := _Broadcast.iSignal[i]._Start;
			IF _nNewStart <> 0 AND_THEN _nNewStart < _nFirstId THEN
				_nFirstId := _Broadcast.iSignal[i]._Start;
				_Broadcast.iFirst := _Broadcast.iSignal[i];
			END_IF
		END_FOR
	END_IF

ELSE
	// 6) Otherwise, swap-remove from the last receiver slot
	_Broadcast.entry[_nPos] := _Broadcast.entry[_nEnd];
	iSignal._End := _nEnd - 1;
END_IF

// 7) Return success code
_Unpair := Ok;

END_FUNCTION

// ---- Entity/Core/Component.TcPOU
(*
Allows registration of FB implementing `I_Component`. The framework will automatically add this function block to the entity's scope.
*)
FUNCTION_BLOCK FINAL Component IMPLEMENTS I_Component
VAR
	_iComponent: I_RawComponent;
	_iEntity: I_Entity;
	_iNext: I_Component;
	_iPrev: I_Component;			
END_VAR

PROPERTY _AsiComponent : I_Component
GET
_AsIComponent := THIS^;
END_GET
END_PROPERTY

PROPERTY _Entity : I_Entity
GET
_Entity := _iEntity;
END_GET
SET
_iEntity := _Entity;
END_SET
END_PROPERTY

PROPERTY _Next : I_ComponentNode
GET
_Next := _iNext;
END_GET
SET
_iNext := _Next._AsiComponent;
END_SET
END_PROPERTY

PROPERTY _Prev : I_ComponentNode
GET
_Prev := _iPrev;
END_GET
SET
_iPrev := _Prev._AsiComponent;
END_SET
END_PROPERTY

(*
Returns parent Entity.
*)
PROPERTY Entity : I_Entity
GET
Entity := _iEntity;
END_GET
END_PROPERTY

//FB_Init is always available implicitly and it is used primarily for initialization.
//The return value is not evaluated. For a specific influence, you can also declare the
//methods explicitly and provide additional code there with the standard initialization
//code. You can evaluate the return value.
{attribute 'hide'}
METHOD FB_init: BOOL
VAR_INPUT
    bInitRetains: BOOL; // TRUE: the retain variables are initialized (reset warm / reset cold)
    bInCopyCode: BOOL;  // TRUE: the instance will be copied to the copy code afterward (online change)
	
	iComponent		: I_RawComponent;
END_VAR
VAR
	_nResult		: Result;
END_VAR
_iComponent := iComponent;

IF _Ec.iUnderConstruction = 0 THEN
	DebugMsg(THIS^, 'Declared outside Entity scope!');
	RETURN;
END_IF
			
IF IsErr(_RegisterComponent(THIS^), nOut => _nResult) THEN
	DebugMsg(THIS^, Tc2_Standard.CONCAT('Failed with code: ', ResultToStr(_nResult)));
END_IF
END_METHOD

(*
Returns raw I_Component pointer.
*)
PROPERTY Raw : I_RawComponent
GET
Raw := _iComponent;
END_GET
END_PROPERTY

END_FUNCTION_BLOCK

// ---- Result/ResultToStr.TcPOU
// Converts a Result value to its corresponding string representation.
// Returns a string that describes the given Result value.
FUNCTION ResultToStr : Str
VAR_INPUT
    nResult : Result; // Result variable to convert to a string
END_VAR

CASE nResult OF
    1: ResultToStr := 'Ok';
    0: ResultToStr := 'None';
    -1: ResultToStr := 'Error';
    -2: ResultToStr := 'Itf0';
    -3: ResultToStr := 'Str0';
    -4: ResultToStr := 'ItfEq';
    -5: ResultToStr := 'NoMatch';
    -6: ResultToStr := 'Ptr0';
    -7: ResultToStr := 'InvRef';
    -8: ResultToStr := 'Ovf';
    -9: ResultToStr := 'Udf';
    -10: ResultToStr := 'Idx';
    -11: ResultToStr := 'TcLib';
    -12: ResultToStr := 'InfLoop';
    -13: ResultToStr := 'IncArg';
	-14: ResultToStr := 'Init';
	-15: ResultToStr := 'Item not found';
	-16: ResultToStr := 'InvItf';
    ELSE
        ResultToStr := Tc2_Standard.CONCAT('Unknown result: ', INT_TO_STRING(nResult));
END_CASE

END_FUNCTION

// ---- Entity/Core/Scope/EntityStart.TcPOU
(*
Represents a registered entity in the Entity-Component system and start of its scope.
Nested scopes are possible, components are always registered within most inner scope.
*)
FUNCTION_BLOCK EntityStart IMPLEMENTS I_Entity, I_Debug;
VAR
	_eState: _EntityState;
	_iNext: I_EntityNode;
	_iPrev: I_EntityNode;
	_iFirstComp: I_Component;
	_iLastComp: I_Component;
	_nSize: UDINT;
END_VAR

PROPERTY INTERNAL _AsIEntity : I_Entity
GET
_AsIEntity := THIS^;
END_GET
END_PROPERTY

PROPERTY INTERNAL _FirstComp : I_ComponentNode
GET
_FirstComp := _iFirstComp;
END_GET
SET
_iFirstComp := _FirstComp._AsiComponent;
END_SET
END_PROPERTY

PROPERTY INTERNAL _LastComp : I_ComponentNode
GET
_LastComp := _iLastComp;
END_GET
SET
_iLastComp := _LastComp._AsiComponent;
END_SET
END_PROPERTY

PROPERTY INTERNAL _Next : I_EntityNode
GET
_Next := _iNext;
END_GET
SET
_iNext := _Next;
END_SET
END_PROPERTY

PROPERTY INTERNAL _Prev : I_EntityNode
GET
_Prev := _iPrev;
END_GET
SET
_iPrev := _Prev;
END_SET
END_PROPERTY

PROPERTY INTERNAL _Size : UDINT
GET
_Size := _nSize;
END_GET
SET
_nSize := _Size;
END_SET
END_PROPERTY

PROPERTY INTERNAL _State : _EntityState
GET
_State := _eState;
END_GET
SET
_eState := _State;
END_SET
END_PROPERTY

//FB_Init is always available implicitly and it is used primarily for initialization.
//The return value is not evaluated. For a specific influence, you can also declare the
//methods explicitly and provide additional code there with the standard initialization
//code. You can evaluate the return value.
{attribute 'hide'}
METHOD FB_Init: BOOL
VAR_INPUT
    bInitRetains: BOOL; // TRUE: the retain variables are initialized (reset warm / reset cold)
    bInCopyCode: BOOL;  // TRUE: the instance will be copied to the copy code afterward (online change)
END_VAR
VAR
	_nResult	: Result;
END_VAR
IF IsErr(_EntityStart(THIS^), nOut => _nResult) THEN
	DebugMsg(THIS^, Tc2_Standard.CONCAT('_StartEntity(THIS^) failed with code: ', ResultToStr(_nResult)));
END_IF
END_METHOD

(*
Retrieves a specific component from the entity based on the provided index.  
Returns `Err.NotFound` if the index is out of range or the entity size is zero.
Returns `Err.InvRef` if the reference to interface variable is invalid.
Otherwise returns `Ok`.
*)
METHOD GetNextComp : Result
VAR_INPUT
	iOut	: REFERENCE TO I_Component;
END_VAR
VAR
	_iThis: I_Entity := THIS^;
END_VAR
// Check if the given output reference is valid
IF NOT __ISVALIDREF(iOut) THEN
    // If not a valid reference, return invalid reference error
    GetNextComp := Err.InvRef;
    RETURN;
END_IF

// If no starting component is specified, begin with the first component
IF iOut = 0 THEN
    IF _iFirstComp <> 0 THEN
        // Return the first component in the list
        iOut := _iFirstComp;
        GetNextComp := Ok;
    ELSE
        // No components exist in the list
        GetNextComp := Err.NotFound;
    END_IF

// If the current component does not belong to this entity, reject the call
ELSIF iOut._Entity <> _iThis THEN
    // Cross-linked or stale reference: component doesn't belong to this context
    GetNextComp := Err.ItfEq;

// If there's no next component, we've reached the end of the list
ELSIF iOut._Next = 0 THEN
    GetNextComp := Err.End;

// Otherwise, return the next component in the list
ELSE
    iOut := iOut._Next._AsiComponent;
    GetNextComp := Ok;
END_IF
END_METHOD

(*
Retrieves a specific component from the entity based on the provided index.  
Returns `Err.NotFound` if the index is out of range or the entity size is zero.
Returns `Err.InvRef` if the reference to interface variable is invalid.
Otherwise returns `Ok`.
*)
METHOD GetPrevComp : Result
VAR_INPUT
	iOut	: REFERENCE TO I_Component;
END_VAR
VAR
	_iThis: I_Entity := THIS^;
END_VAR
// Check if the given output reference is valid
IF NOT __ISVALIDREF(iOut) THEN
    // If not a valid reference, return invalid reference error
    GetPrevComp := Err.InvRef;
    RETURN;
END_IF

// If no starting component is specified, begin with the first component
IF iOut = 0 THEN
    IF _iLastComp <> 0 THEN
        // Return the first component in the list
        iOut := _iLastComp;
        GetPrevComp := Ok;
    ELSE
        // No components exist in the list
        GetPrevComp := Err.NotFound;
    END_IF

// If the current component does not belong to this entity, reject the call
ELSIF iOut._Entity <> _iThis THEN
    // Cross-linked or stale reference: component doesn't belong to this context
    GetPrevComp := Err.ItfEq;

// If there's no next component, we've reached the end of the list
ELSIF iOut._Prev = 0 THEN
    GetPrevComp := Err.End;

// Otherwise, return the next component in the list
ELSE
    iOut := iOut._Prev._AsiComponent;
    GetPrevComp := Ok;
END_IF
END_METHOD

(*
Provides the size of the entity, indicating the number of components it manages.  
Note: For internal logic purposes, this value is incremented by one beyond the actual component count.
*)
PROPERTY Size : UDINT
GET
Size := _nSize;
END_GET
END_PROPERTY

END_FUNCTION_BLOCK

// ---- Entity/Sys/_Helpers/_EntityStart.TcPOU
FUNCTION INTERNAL _EntityStart : Result
VAR_INPUT
	iEntity: I_Entity;
END_VAR

// Check if the runtime system has been initialized
IF NOT _Runtime.bInit THEN
    // If not initialized, return with an initialization error
    _EntityStart := Err.Init;
    RETURN;
END_IF

// Check if the input entity reference is valid
IF iEntity = 0 THEN
    // If invalid, return with interface error
    _EntityStart := Err.Itf0;
    RETURN;
END_IF

// Ensure the entity is in the 'Unregistered' state before registering
IF iEntity._State <> _EntityState.Unregistered THEN
    // If already registered or in an unexpected state, return error
    _EntityStart := Err.ItfEq;
    RETURN;
END_IF

// If this is the first entity in the scope, initialize the list
IF _Ec.iLast = 0 THEN
    _Ec.iFirst := iEntity;       // Set as first entity
    _Ec.iLast := iEntity;        // Set as last entity
ELSE
    // Link the new entity to the end of the current list						| iOther < iLast > 0			| 0 < iEntity > 0 
    _Ec.iLast._Next := iEntity;  // Set previous last's next to new entity		| iOther < iLast > iEntity		| 0 < iEntity > 0
    iEntity._Prev := _Ec.iLast;  // Set new entity's previous to old last		| iOther < iLast > iEntity		| iLast < iEntity > 0
    _Ec.iLast := iEntity;        // Update the last entity pointer				| iLast = iEntity
END_IF

// Register the entity and prepare for construction
iEntity._State := _EntityState.Registered;
_Ec.iUnderConstruction := iEntity;

// Increment the scope construction count
_Ec.nConstructedScopes := _Ec.nConstructedScopes + 1;
_EntityStart := Ok;

END_FUNCTION

// ---- Entity/Core/GetOwnerFromRaw.TcPOU
(*
Finds the owning entity of a given component in the Entity-Component system.  
This function may involve a costly search operation, iterating through all components.
Returns:
- `Ok` - Successfully retrieves the `I_Entity` that owns the component.
- `Err.Itf0` - iIn = 0.
- `Err.InvRef` - Invalid output reference.
- `Err.NotFound` - No owning entity is found, returning null.
*)
FUNCTION GetOwnerFromRaw : Result
VAR_INPUT
	iIn: I_Component;
	iOut: REFERENCE TO I_Entity;
END_VAR
VAR
	i			: Iter(1);
	j			: Iter(1);
	_iComp		: I_FatComponent;
END_VAR

IF iIn = 0 THEN
	GetOwnerFromRaw := Err.Itf0;
	RETURN;
END_IF

IF NOT __ISVALIDREF(iOut) THEN
	GetOwnerFromRaw := Err.InvRef;
	RETURN;
END_IF

WHILE IsOk(GetEntity(i.Next(), iOut)) DO
	j.Set(1);
	WHILE IsOk(iOut.Get(j.Next(), _iComp)) DO
		IF _iComp.Raw = iIn THEN
			GetOwnerFromRaw := Ok;
			RETURN;
		END_IF
	END_WHILE
END_WHILE

GetOwnerFromRaw := Err.NotFound;

END_FUNCTION

// ---- Iter/Iter.TcPOU
// Provides iteration functionality over UDINT value.
// Requires initialization value.
FUNCTION_BLOCK FINAL Iter
VAR
	_nIter		: UDINT;
	_bFirstLoop	: BOOL := TRUE;
END_VAR

//FB_Init is always available implicitly and it is used primarily for initialization.
//The return value is not evaluated. For a specific influence, you can also declare the
//methods explicitly and provide additional code there with the standard initialization
//code. You can evaluate the return value.
{attribute 'hide'}
METHOD FB_Init: BOOL
VAR_INPUT
    bInitRetains: BOOL; // TRUE: the retain variables are initialized (reset warm / reset cold)
    bInCopyCode: BOOL;  // TRUE: the instance will be copied to the copy code afterward (online change)

	nInit		: UDINT; // Sets the initial iteration value to nInit.
END_VAR
_nIter := nInit;
END_METHOD

// Returns the current iteration value.
METHOD Get : UDINT
VAR_INPUT
END_VAR
Get := _nIter;
END_METHOD

// Increments the iteration value unless it's the first loop.
// On the first loop, returns the initial value without incrementing.
METHOD Next : UDINT
VAR_INPUT
END_VAR
IF _bFirstLoop THEN
	_bFirstLoop := FALSE;
	Next := _nIter;
	RETURN;	
END_IF

_nIter := _nIter + 1;
Next := _nIter;
END_METHOD

// Returns the next iteration value without modifying the current state.
METHOD Peek: UDINT
VAR_INPUT
END_VAR
Peek := _nIter + 1;
END_METHOD

// Returns the previous iteration value without modifying the current state.
METHOD PeekBack: UDINT
VAR_INPUT
END_VAR
PeekBack := _nIter - 1;
END_METHOD

// Decrements the iteration value unless it's the first loop.
// On the first loop, returns the initial value without decrementing.
METHOD Prev: UDINT
VAR_INPUT
END_VAR
IF _bFirstLoop THEN
	_bFirstLoop := FALSE;
	Prev := _nIter;
	RETURN;	
END_IF

_nIter := _nIter - 1;
Prev := _nIter;
END_METHOD

// Sets the iteration to a new value and resets the first loop flag.
// Returns the new value of the iteration.
METHOD Set: UDINT
VAR_INPUT
    nNewValue: UDINT; // New value to set for the iteration
END_VAR
_nIter := nNewValue;
_bFirstLoop	:= TRUE;
Set := _nIter;
END_METHOD

END_FUNCTION_BLOCK

// ---- Entity/Core/GetNextEntity.TcPOU
(*
Retrieves the I_Entity instance. It is either next entity in relation to the inputted one or first entity if passed interface pointer contains null.

Results:
- Ok - Success. Replaces value of iEntity with the first or following entity.
- Err.InvRef - Invalid reference.
- Err.Itf0 - No entity. Nulls passed interface pointer.
- Err.End - End of collection. Nulls passed interface pointer.
*)
FUNCTION GetNextEntity : Result
VAR_INPUT
	iEntity: REFERENCE TO I_Entity;
END_VAR
VAR
END_VAR

// Check if the given entity reference is valid
IF NOT __ISVALIDREF(iEntity) THEN
    // If the reference is invalid, return with an invalid reference error
    GetNextEntity := Err.InvRef;
    RETURN;
END_IF

// Check if the entity chain has been initialized (i.e., if there's a first entity)
IF _Ec.iFirst = 0 THEN
    // If not initialized, return with interface error
	iEntity := 0;
    GetNextEntity := Err.Itf0;
    RETURN;
END_IF

// If input entity is 0, start iteration from the first entity in the list
IF iEntity = 0 THEN
    iEntity := _Ec.iFirst._AsIEntity;
    GetNextEntity := Ok;

// If the current entity has a next one, move to it
ELSIF iEntity._Next <> 0 THEN
    iEntity := iEntity._Next._AsIEntity;
    GetNextEntity := Ok;

// If there is no next entity, end of the list is reached
ELSE
    iEntity := 0;
    GetNextEntity := Err.End;
END_IF

END_FUNCTION

// ---- Entity/Core/GetPrevEntity.TcPOU
(*
Retrieves the I_Entity instance. It is either previous entity in relation to the inputted one or last entity if passed interface pointer contains null.

Results:
- Ok - Success. Replaces value of iEntity with the last or previous entity.
- Err.InvRef - Invalid reference.
- Err.Itf0 - No entity. Nulls passed interface pointer.
- Err.End - End of collection. Nulls passed interface pointer.
*)
FUNCTION GetPrevEntity : Result
VAR_INPUT
	iEntity: REFERENCE TO I_Entity;
END_VAR
VAR
END_VAR

// Check if the given entity reference is valid
IF NOT __ISVALIDREF(iEntity) THEN
    // If the reference is invalid, return with an invalid reference error
    GetPrevEntity := Err.InvRef;
    RETURN;
END_IF

// Check if the entity chain has been initialized (i.e., if there's a last entity)
IF _Ec.iLast = 0 THEN
    // If not initialized, return with interface error
	iEntity := 0;
    GetPrevEntity := Err.Itf0;
    RETURN;
END_IF

// If input entity is 0, start iteration from the last entity in the list
IF iEntity = 0 THEN
    iEntity := _Ec.iLast._AsIEntity;
    GetPrevEntity := Ok;

// If the current entity has a previous one, move to it
ELSIF iEntity._Prev <> 0 THEN
    iEntity := iEntity._Prev._AsIEntity;
    GetPrevEntity := Ok;

// If there is no previous entity, beginning of the list is reached
ELSE
	iEntity := 0;
    GetPrevEntity := Err.End;
END_IF

END_FUNCTION

// ---- Entity/Sys/_Helpers/_EntityExtend.TcPOU
FUNCTION INTERNAL _EntityExtend : Result
VAR_INPUT
	iEntity	: I_Entity;
END_VAR

// Check if the runtime system has been initialized
IF NOT _Runtime.bInit THEN
    // If not initialized, return with an initialization error
    _EntityExtend := Err.Init;
    RETURN;
END_IF

// Check if the provided entity reference is valid
IF iEntity = 0 THEN
    // If invalid, return with interface error
    _EntityExtend := Err.Itf0;
    RETURN;
END_IF

// Ensure the entity is in the 'Completed' state before proceeding
IF iEntity._State <> _EntityState.Completed THEN
    // If not completed, return with incorrect argument error
    _EntityExtend := Err.IncArg;
    RETURN;
END_IF

// Mark the entity as 'Registered' for extension
iEntity._State := _EntityState.Registered;

// Set the entity as the current one under construction
_Ec.iUnderConstruction := iEntity;

// Increment the scope construction counter
_Ec.nConstructedScopes := _Ec.nConstructedScopes + 1;
_EntityExtend := Ok;

END_FUNCTION

// ---- Result/IsEnd.TcPOU
// Return TRUE for any value other than None (0).
// Optionally carries the value over to nOut for further processing.
FUNCTION IsEnd : BOOL
VAR_INPUT
    nIn : Result; // Result variable to check for any non-None value
END_VAR
VAR_OUTPUT
    nOut : Result; // Carries the input value for further use
END_VAR

IsEnd := nIn = Err.End;
nOut := nIn;

END_FUNCTION

// ---- Runtime/Runtime.TcPOU
(*
Manages the initialization and cyclic execution of registered function blocks.
*)
FUNCTION Runtime
VAR
	iInit: I_InitNode := _Runtime.iFirstInit;
	iExecute: I_ExecuteNode := _Runtime.iFirstCyclic;
END_VAR

IF _Runtime.bInit THEN
	WHILE iInit <> 0 DO
		iInit.Init(iNext => iInit);
	END_WHILE

	IF _Ec.nConstructedScopes <> 0 THEN
		DebugMsg(0, 'Close all Entity scopes!');
	END_IF
	
	IF _Debug.nErrorNumber > 0 THEN
		_Runtime.iFirstCyclic := 0;
		Tc2_System.ADSLOGSTR(Tc2_System.ADSLOG_MSGTYPE_ERROR, Tc2_Standard.CONCAT('Runtime disabled! Errors: ', UDINT_TO_STRING(_Debug.nErrorNumber)), '');
	END_IF
	
	_Runtime.bInit := FALSE;
END_IF

WHILE iExecute <> 0 DO
	iExecute.Exe(iNext => iExecute);
END_WHILE

END_FUNCTION

// ---- State/Helpers/GetStateManager.TcPOU
(*
Searches an `I_Entity` for a `I_StateManager` component matching provided id pattern.
Result:
- Ok - Returns `I_StateManager`.
- Err.NotFound - Returns null.
- Err.InvRef - Returns null.
- Err.Itf0 - Returns null, incorrect interface.
*)
FUNCTION GetStateManager : Result
VAR_INPUT
	iEntity		: I_Entity;
	iOut		: REFERENCE TO I_StateManager;
END_VAR
VAR
	i			: Iter(1);
	_iComp		: I_FatComponent;
	cmp			: TagCmp;
END_VAR

IF iEntity = 0 THEN
	GetStateManager := Err.Itf0;
	RETURN;
END_IF

IF NOT __ISVALIDREF(iOut) THEN
	GetStateManager := Err.InvRef;
	RETURN;
END_IF

WHILE IsOk(iEntity.Get(i.Next(), _iComp)) DO
	IF IsOk(ICompToIStateMgr(_iComp.Raw, iOut)) THEN
		GetStateManager := Ok;
		RETURN;
	END_IF
END_WHILE

GetStateManager := Err.NotFound;

END_FUNCTION

// ---- State/Helpers/GetState.TcPOU
(*
Searches an `I_Entity` for a `I_State` component matching provided id pattern.
Result:
- Ok - Returns `I_State`.
- Err.NotFound - Returns null.
- Err.InvRef - Returns null.
- Err.Itf0 - Returns null, incorrect interface.
*)
FUNCTION GetState : Result
VAR_INPUT
	iEntity		: I_Entity;
	sTagId		: Str;
	iOut		: REFERENCE TO I_State;
END_VAR
VAR
	_iComp		: I_Component;
	cmp			: TagCmp;
END_VAR

IF iEntity = 0 THEN
	GetState := Err.Itf0;
	RETURN;
END_IF

IF NOT __ISVALIDREF(iOut) THEN
	GetState := Err.InvRef;
	RETURN;
END_IF

WHILE IsOk(iEntity.GetNextComp(_iComp)) DO
	IF IsOk(ICompToIState(_iComp.Raw, iOut)) THEN
		IF cmp.Set(iOut.Tag).MatchWcdId(sTagId).IsTrue() THEN
			GetState := Ok;
			RETURN;
		ELSE
			iOut := 0;
		END_IF
	END_IF
END_WHILE

GetState := Err.NotFound;

END_FUNCTION

// ---- State/State/ICompToIState.TcPOU
(*
Casts I_Component as I_State.
Returns:
- Ok - Success,
- Err.InvRef - Invalid reference,
- Err.Itf0 - Invalid interface,
- Err.NoMatch - Cast failed
*)
FUNCTION ICompToIState : Result
VAR_INPUT
	iIn		: I_RawComponent;
	iOut	: REFERENCE TO I_State;
END_VAR

IF NOT __ISVALIDREF(iOut) THEN
	ICompToIState := Err.InvRef;
	RETURN;
END_IF

IF iIn = 0 THEN
	ICompToIState := Err.Itf0;
	RETURN;
END_IF

IF __QUERYINTERFACE(iIn, iOut) THEN
	ICompToIState := Ok;
ELSE
	ICompToIState := Err.NoMatch;
END_IF

END_FUNCTION

// ---- Tags/Casts/ICompToITag.TcPOU
(*
Casts I_Component as I_Tag.
Returns:
- Ok - Success,
- Err.InvRef - Invalid reference,
- Err.Itf0 - Invalid interface,
- Err.NoMatch - Cast failed
*)
FUNCTION ICompToITag : Result
VAR_INPUT
	iIn		: I_RawComponent;
	iOut	: REFERENCE TO I_Tag;
END_VAR

IF NOT __ISVALIDREF(iOut) THEN
	ICompToITag := Err.InvRef;
	RETURN;
END_IF

IF iIn = 0 THEN
	ICompToITag := Err.Itf0;
	RETURN;
END_IF

IF __QUERYINTERFACE(iIn, iOut) THEN
	ICompToITag := Ok;
ELSE
	ICompToITag := Err.NoMatch;
END_IF

END_FUNCTION

// ---- Tags/Casts/ICompToITagged.TcPOU
(*
Casts I_Component as I_Tagged.
Returns:
- Ok - Success,
- Err.InvRef - Invalid reference,
- Err.Itf0 - Invalid interface,
- Err.NoMatch - Cast failed
*)
FUNCTION ICompToITagged : Result
VAR_INPUT
	iIn		: I_RawComponent;
	iOut	: REFERENCE TO I_Tagged;
END_VAR

IF NOT __ISVALIDREF(iOut) THEN
	ICompToITagged := Err.InvRef;
	RETURN;
END_IF

IF iIn = 0 THEN
	ICompToITagged := Err.Itf0;
	RETURN;
END_IF

IF __QUERYINTERFACE(iIn, iOut) THEN
	ICompToITagged := Ok;
ELSE
	ICompToITagged := Err.NoMatch;
END_IF

END_FUNCTION

// ---- Tags/Helpers/GetTagOption.TcPOU
(*
Searches an `I_Entity` for a `I_Tag` component with provided `Option` value.
Result:
- Ok - Returns iTag.
- Err.NotFound - Returns null.
- Err.InvRef - Provided reference is invalid.
- Err.Itf0 - Returns null, incorrect interface.
*)
FUNCTION GetTagOption : Result
VAR_INPUT
	iEntity		: I_Entity;
	sOption		: Str;
	iOut		: REFERENCE TO I_Tag;
END_VAR
VAR
	i			: Iter(1);
	_iComp		: I_FatComponent;
END_VAR

IF iEntity = 0 THEN
	GetTagOption := Err.Itf0;
	RETURN;
END_IF

IF NOT __ISVALIDREF(iOut) THEN
	GetTagOption := Err.InvRef;
	RETURN;
END_IF

WHILE IsOk(iEntity.Get(i.Next(), _iComp)) DO
	IF IsOk(ICompToITag(_iComp.Raw, iOut)) THEN
		IF iOut.Option = sOption THEN
			GetTagOption := Ok;
			RETURN;
		ELSE
			iOut := 0;
		END_IF
	END_IF
END_WHILE

GetTagOption := Err.NotFound;

END_FUNCTION

// ---- Tags/Helpers/HasTag.TcPOU
(*
Searches an `I_Entity` for a `I_Tag` component matching provided id pattern.
Result:
- Ok
- Err.NotFound - Returns null.
- Err.Itf0 - Returns null, incorrect interface.
*)
FUNCTION HasTag : Result
VAR_INPUT
	iEntity		: I_Entity;
	sIdPattern	: Str;
END_VAR
VAR
	_iComp		: I_Component;
	_iTag		: I_Tag;
	cmp			: TagCmp;
END_VAR

IF iEntity = 0 THEN
	HasTag := Err.Itf0;
	RETURN;
END_IF

WHILE IsOk(iEntity.GetNextComp(_iComp)) DO
	IF IsOk(ICompToITag(_iComp.Raw, _iTag)) THEN
		IF cmp.Set(_iTag).MatchWcdId(sIdPattern).IsTrue() THEN
			HasTag := Ok;
			RETURN;
		END_IF
	END_IF
END_WHILE

HasTag := Err.NotFound;

END_FUNCTION
